(* PLC project Sem nome, Desconhecido Sem nome 1 *)
(* stored: creationDateTime 2023-06-20T14:48:23, modificationDateTime 2023-06-20T20:08:32 *)

PROGRAM program0

            PROGRAM ON_OFF_Controller

VAR

    setpoint: REAL := 25.0;  // Valor de referência desejado

    hysteresis: REAL := 1.0; // Histerese para evitar oscilações

    output: BOOL := FALSE;   // Saída do controlador

    input: REAL;             // Valor da entrada

END_VAR



METHOD Controlador_ON_OFF : BOOL

VAR

    error: REAL;  // Erro entre o setpoint e o valor de entrada

BEGIN

    error := input - setpoint;  // Calcula o erro

    

    IF error > hysteresis THEN

        output := TRUE;   // Liga a saída se o erro for maior que a histerese

    ELSIF error < -hysteresis THEN

        output := FALSE;  // Desliga a saída se o erro for menor que a histerese

    END_IF;

    

    RETURN output;  // Retorna o valor da saída

END_METHOD


          
END_PROGRAM

CONFIGURATION Config0
  RESOURCE Res0 ON PLC
    TASK task0(INTERVAL := T#20ms, PRIORITY := 0);
    PROGRAM instance0 WITH task0 : program0;
  END_RESOURCE
END_CONFIGURATION
